{attribute 'GeneratedUsingTerminal: EL6002-0000-0017'}
{attribute addProperty BoxType "EL6002-0000-0017"}
{attribute addProperty Id "EtcSlaveTerminalBaseCOM_TxPDO_Map_Inputs_Channel_1AT %I*COM_TxPDO_Map_Inputs_Channel_3801C95E30COM_TxPDO_Map_Inputs_Channel_2AT %I*COM_TxPDO_Map_Inputs_Channel_3801C95E30COM_RxPDO_Map_Outputs_Channel_1AT %Q*COM_RxPDO_Map_Outputs_Channel_EADA2E0D27COM_RxPDO_Map_Outputs_Channel_2AT %Q*COM_RxPDO_Map_Outputs_Channel_EADA2E0D27WcStateAT %I*WcState_9091E0EB2InfoDataAT %I*InfoData_32EB74EA10"}
{attribute addProperty CRC "341417789"}
{attribute addProperty Size "126"}
TYPE EL6002_14599F3D EXTENDS EtcSlaveTerminalBase :
STRUCT
	{attribute addProperty Name "COM_TxPDO_Map_Inputs_Channel_1"}
	COM_TxPDO_Map_Inputs_Channel_1 : COM_TxPDO_Map_Inputs_Channel_3801C95E;
	{attribute addProperty Name "COM_TxPDO_Map_Inputs_Channel_2"}
	COM_TxPDO_Map_Inputs_Channel_2 : COM_TxPDO_Map_Inputs_Channel_3801C95E;
	{attribute addProperty Name "COM_RxPDO_Map_Outputs_Channel_1"}
	COM_RxPDO_Map_Outputs_Channel_1 : COM_RxPDO_Map_Outputs_Channel_EADA2E0D;
	{attribute addProperty Name "COM_RxPDO_Map_Outputs_Channel_2"}
	COM_RxPDO_Map_Outputs_Channel_2 : COM_RxPDO_Map_Outputs_Channel_EADA2E0D;
	{attribute addProperty Name "WcState"}
	WcState : WcState_9091E0EB;
	{attribute addProperty Name "InfoData"}
	InfoData : InfoData_32EB74EA;
END_STRUCT
END_TYPE

(* stored: Version 1.2.0.0, ProductVersion 3.1.4024.9
   DUT EL6002_14599F3D: Id {06b13d60-39ae-4858-9f29-548e6de19e8c} *)
